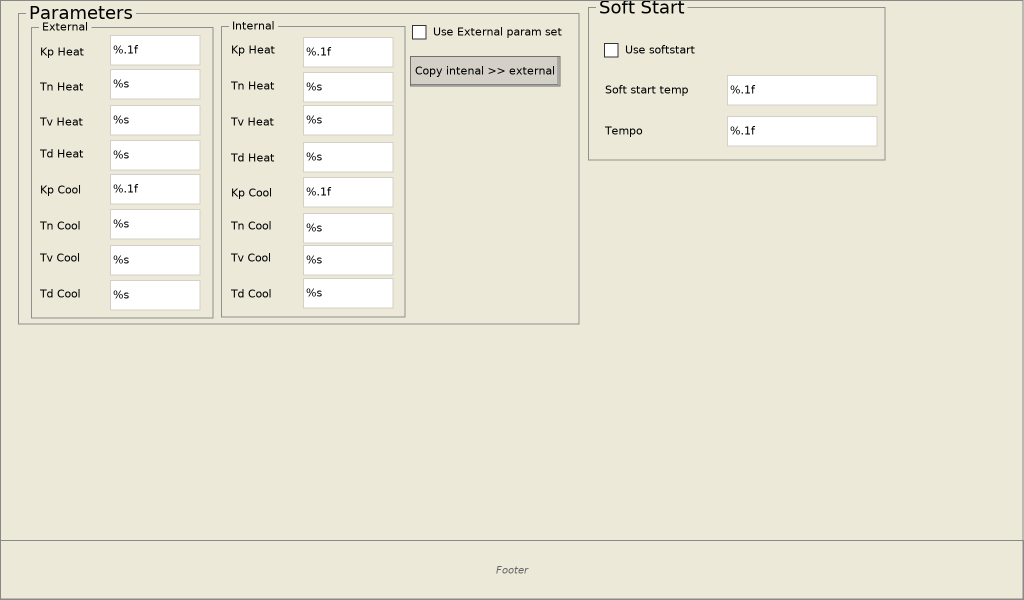
VISUALIZATION ExtraParams  // 1024x600
    GroupBox (18,5 561x319), "Parameters"
        GroupBox (13,14 182x299), "External"
            Label (6,18 70x30), "Kp Heat"
            Label (6,53 70x30), "Tn Heat"
            Label (6,88 70x30), "Tv Heat"
            Label (6,120 70x30), "Td Heat"
            Label (6,156 70x30), "Kp Cool"
            Label (6,192 70x30), "Tn Cool"
            Label (6,224 70x30), "Tv Cool"
            Label (6,260 70x30), "Td Cool"
            Textfield (79,16 90x30), "%.1f", text variable: MAIN.externalParams.KpHeat
            Textfield (79,50 90x30), "%s", text variable: MAIN.externalParams.TnHeat
            Textfield (79,86 90x30), "%s", text variable: MAIN.externalParams.TvHeat
            Textfield (79,121 90x30), "%s", text variable: MAIN.externalParams.TdHeat
            Textfield (79,155 90x30), "%.1f", text variable: MAIN.externalParams.KpCool
            Textfield (79,190 90x30), "%s", text variable: MAIN.externalParams.TnCool
            Textfield (79,226 90x30), "%s", text variable: MAIN.externalParams.TvCool
            Textfield (79,261 90x30), "%s", text variable: MAIN.externalParams.TdCool
        GroupBox (203,13 184x299), "Internal"
            Label (7,17 70x30), "Kp Heat"
            Label (7,53 70x30), "Tn Heat"
            Label (7,89 70x30), "Tv Heat"
            Label (7,125 70x30), "Td Heat"
            Label (7,160 70x30), "Kp Cool"
            Label (7,193 70x30), "Tn Cool"
            Label (7,225 70x30), "Tv Cool"
            Label (7,261 70x30), "Td Cool"
            Textfield (82,19 90x30), "%.1f", text variable: MAIN.internalParams.KpHeat
            Textfield (82,54 90x30), "%s", text variable: MAIN.internalParams.TnHeat
            Textfield (82,87 90x30), "%s", text variable: MAIN.internalParams.TvHeat
            Textfield (82,124 90x30), "%s", text variable: MAIN.internalParams.TdHeat
            Textfield (82,159 90x30), "%.1f", text variable: MAIN.internalParams.KpCool
            Textfield (82,195 90x30), "%s", text variable: MAIN.internalParams.TnCool
            Textfield (82,227 90x30), "%s", text variable: MAIN.internalParams.TvCool
            Textfield (82,260 90x30), "%s", text variable: MAIN.internalParams.TdCool
        Checkbox (392,12 172x30), "Use External param set", tooltip "When activated select the external params", variable: MAIN.stControllerParameter.bSelCtrlParameterSet
        Button (392,51 150x30), "Copy intenal >> external"
            tap MAIN.bCopyParams
    Frame (0,540 1024x60)
        shows Footer()
    GroupBox (588,-1 297x161), "Soft Start"
        Checkbox (14,36 116x30), "Use softstart", variable: MAIN.stControllerParameter.bEnableSoftStart
        Label (14,76 116x30), "Soft start temp"
        Textfield (139,76 150x30), "%.1f", text variable: MAIN.stControllerParameter.fWStartUp
            OnMouseClick: write the text variable via Default
        Label (14,117 100x30), "Tempo"
        Textfield (139,117 150x30), "%.1f", text variable: MAIN.softStartWaitTime
            OnMouseClick: write the text variable via Default
END_VISUALIZATION

(* stored: Version 1.1.0.1, ProductVersion 3.1.4024.12
   Visu ExtraParams: Id {d0e8b4ae-d5ed-4589-a274-36ff51b2e552} *)
